// TIA Portal project "uMySQL_V0.3" (V15.1)

(* hardware
DEVICE "S7-1200 station_1"  S7-1200 Station
   slot 0: "Rack_0"  S7-1200 Rack  Rack  V1.0
   slot 1: "PLC_1"  CPU 1215C DC/DC/DC  6ES7 215-1AG40-0XB0  V4.2
*)

// ===== PLC "PLC_1"  CPU 1215C DC/DC/DC =====

VAR_GLOBAL   // PLC tag table "默认变量表"
   "Tag_1" AT %M100.0 : Bool;
   "Tag_2" AT %M100.1 : Bool;
   "Tag_3" AT %M100.2 : Bool;
END_VAR

TYPE "uMySQL_CDD"
   STRUCT
      Connect_OK : Bool;
      Connect_ID : Conn_Ouc;
      Connect_Sequence : DInt;
      Server_Protocol_Version : Int;
      Server_Server_Version : String;
      Server_Character_Set : Byte;
      CLIENT_PLUGIN_AUTH : String;
   END_STRUCT;
END_TYPE

DATA_BLOCK "uMySQL_Connect_DB"   // DB1
{ S7_Optimized_Access := 'TRUE' }
VERSION : 0.1
// stored: InstanceOfName uMySQL_Connect
"uMySQL_Connect"
BEGIN
   IP.RemoteAddress.ADDR[4] := 16#E0;
   IP.InterfaceId := 64;
   IP.ID := 16#65;
END_DATA_BLOCK

DATA_BLOCK "测试数据块"   // DB2
{ S7_Optimized_Access := 'TRUE' }
VERSION : 0.1
   VAR
      wstring : WString[2048];
      ad : Array[0..2048] of Byte;
   END_VAR
BEGIN
END_DATA_BLOCK

DATA_BLOCK "uMySQL_Query_DB"   // DB3
{ S7_Optimized_Access := 'TRUE' }
VERSION : 0.1
// stored: InstanceOfName uMySQL_Query
"uMySQL_Query"
BEGIN
END_DATA_BLOCK

DATA_BLOCK "uMySQL_Query_DB_1"   // DB4
{ S7_Optimized_Access := 'TRUE' }
VERSION : 0.1
// stored: InstanceOfName uMySQL_Query
"uMySQL_Query"
BEGIN
END_DATA_BLOCK

DATA_BLOCK "uMySQL_INI_DB_DB"   // DB5
{ S7_Optimized_Access := 'TRUE' }
VERSION : 0.1
// stored: InstanceOfName uMySQL_INI_DB
"uMySQL_INI_DB"
BEGIN
END_DATA_BLOCK

ORGANIZATION_BLOCK "Main"   // OB1, LAD, ProgramCycle
TITLE = "Main Program Sweep (Cycle)"
{ S7_Optimized_Access := 'TRUE' }
VERSION : 0.1
   VAR_INPUT
      Initial_Call : Bool;   // Initial call of this OB
      Remanence : Bool;   // =True, if remanent data are available
   END_VAR
BEGIN

REGION Network 1
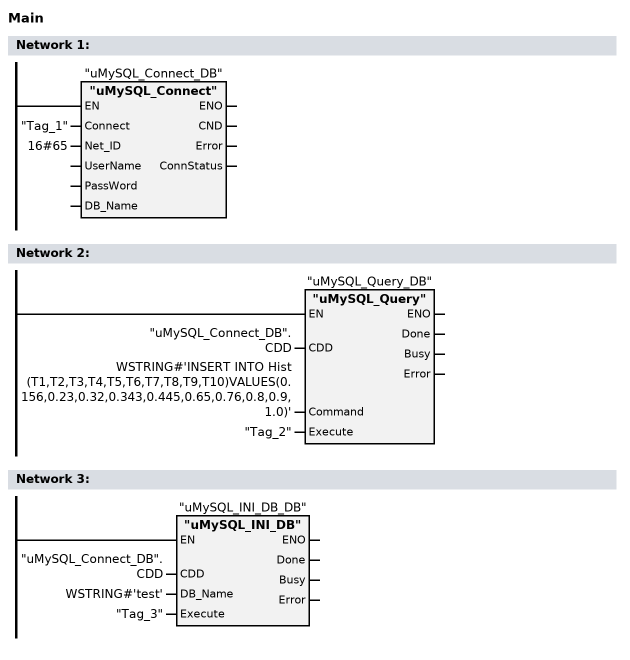
   RUNG wire#powerrail
      "uMySQL_Connect_DB"(Connect := "Tag_1", Net_ID := 16#65, UserName :=, PassWord :=, DB_Name :=, CND =>, Error =>, ConnStatus =>)
   END_RUNG
   // the same network as SCL:
   "uMySQL_Connect_DB"(Connect := "Tag_1", Net_ID := 16#65);   // "uMySQL_Connect"
END_REGION

REGION Network 2
   RUNG wire#powerrail
      "uMySQL_Query_DB"(CDD := "uMySQL_Connect_DB".CDD, Command := WSTRING#'INSERT INTO Hist (T1,T2,T3,T4,T5,T6,T7,T8,T9,T10)VALUES(0.156,0.23,0.32,0.343,0.445,0.65,0.76,0.8,0.9,1.0)', Execute := "Tag_2", Done =>, Busy =>, Error =>)
   END_RUNG
   // the same network as SCL:
   "uMySQL_Query_DB"(CDD := "uMySQL_Connect_DB".CDD,   // "uMySQL_Query"
                     Command := WSTRING#'INSERT INTO Hist (T1,T2,T3,T4,T5,T6,T7,T8,T9,T10)VALUES(0.156,0.23,0.32,0.343,0.445,0.65,0.76,0.8,0.9,1.0)',
                     Execute := "Tag_2");
END_REGION

REGION Network 3
   RUNG wire#powerrail
      "uMySQL_INI_DB_DB"(CDD := "uMySQL_Connect_DB".CDD, DB_Name := WSTRING#'test', Execute := "Tag_3", Done =>, Busy =>, Error =>)
   END_RUNG
   // the same network as SCL:
   "uMySQL_INI_DB_DB"(CDD := "uMySQL_Connect_DB".CDD, DB_Name := WSTRING#'test', Execute := "Tag_3");   // "uMySQL_INI_DB"
END_REGION
END_ORGANIZATION_BLOCK

// folder: uMySQL

FUNCTION_BLOCK "uMySQL_Connect"   // FB3, SCL
{ S7_Optimized_Access := 'TRUE' }
VERSION : 0.1
   VAR_INPUT
      Connect : Bool;   // True:发起连接；False:断开连接
      Net_ID : Conn_Ouc;   // 连接ID
      UserName : String := 'root';   // 数据库用户名
      PassWord : String := 'root';   // 数据库密码
      DB_Name : String := 'hist';   // 数据库名
   END_VAR
   VAR_OUTPUT
      CND : Bool;
      Error : Bool;
      ConnStatus : Byte;
   END_VAR
   VAR
      IP : TCON_IP_v4;
      CDD : "uMySQL_CDD";   // 共用的数据库连接参数
      TempBool : Array[0..19] of Bool;
      REV_Buffer : Array[0..#MessageMaxLen] of Byte;
      SND_Buffer : Array[0..#MessageMaxLen] of Byte;
      NetConnect : TCON;
      NetRcv : TRCV;
      NetRcv_EN : Bool;
      NetRcv_Len : Int;
      NetRcv_Done : Bool;
      "Step" : Int;
      MessageLen : Int;   // 消息帧长度
      SaltLen : Int;   // 挑战随机数长度
      Server_Auth_PlugIn_Name : String;
      ServerVersion_StartNum : Int;
      ServerCapability_flag : DWord;
      SaltString : Array[0..49] of Byte;
      Client_CapabilityFlag : DWord := 16#8609;   // 客户端权能标志位
      Client_MaxLen : DWord;
      Calc_Encryption_SHA1 : "Calc_Encryption_SHA1";
      Temp_SHA1 : Array[0..19] of Byte;
      Temp_SHA_Arry : Array[0..55] of Byte;
      Temp_SHA_Arry_Num : UInt;
      Temp_SHA_Arry_Num_Int : Int;
      Temp_SHA1_2 : Array[0..19] of Byte;
      Temp_SHA1_3 : Array[0..19] of Byte;
      Token : Array[0..19] of Byte;
      NetDISCON : TDISCON;
      NetDiscon_EN : Bool;
      NetSend : TSEND;
      NetSend_EN : Bool;
      NetSend_Done : Bool;
      TDiag_Result : TDiag_Status;
      NetDiag : T_DIAG;
      NetDiag_EN : Bool;
      NetSendLen : Int;
      Timer_ON : TON_TIME;
      Timer_OFF : TON_TIME;
      Timer_Error : TON_TIME;
      NetSendEnd : TSEND;
      NetSendEnd_EN : Bool;
      NetSendEnd_Done : Bool;
   END_VAR
   VAR_TEMP
      Temp_Dword : DWord;
      Temp_Index_i : Int;
      Temp_NowNum : Int;
      Temp_StrLen : Int;
   END_VAR
   VAR CONSTANT
      MessageMaxLen : DInt := 2048;   // 收发消息的最大长度
   END_VAR
   // IP.RemotePort := 3306;
   // IP.RemoteAddress.ADDR[4] := 16#A8;
   // IP.RemoteAddress.ADDR[3] := 16#1F;
   // IP.RemoteAddress.ADDR[2] := 16#A8;
   // IP.RemoteAddress.ADDR[1] := 16#C0;
   // IP.ActiveEstablished := true;
   // // CDD.Connect_OK : 数据库是否连接状态True:已连接；False :未连接
   // // CDD.Connect_ID : 连接ID，用于传递
   // // CDD.Connect_Sequence : 命令Sequence，用于传递
BEGIN


   (***********************************************************初始化数据******************************************************************)
   IF #Connect AND  #TempBool[0]=FALSE THEN
       #TempBool[0] := TRUE;
       #TempBool[1] := FALSE;
       #Step := 0;
       #CDD.Connect_ID := #Net_ID;
       #IP.ID := #Net_ID;
       #NetRcv_EN := TRUE;
       #NetDiscon_EN := FALSE;
       #NetSendEnd_EN := FALSE;
       ;
   END_IF;
   (***********************************************************断开连接******************************************************************)
   IF #Connect = FALSE AND #TempBool[1]=FALSE THEN
       #TempBool[0] := FALSE;
       #TempBool[1] := TRUE;
       #Step := 6;
   END_IF;


   #NetConnect(REQ:=#Connect,
               ID:=  #CDD.Connect_ID,
               CONNECT:=#IP);
   #NetRcv(EN_R:=#NetRcv_EN,
           ID:=#CDD.Connect_ID,
           LEN:=0,
           ADHOC:=TRUE,
           DATA:=#REV_Buffer);
   IF #NetRcv.NDR THEN
       #NetRcv_Done := TRUE;
   END_IF;
   (***********************************************************处理流程******************************************************************)
   //#Step 0  发起连接
   //#Step 1 等待MySQL服务器发回来的数据
   //#Step 2 解码发回来的认证数据，并计算需要响应的数据放入Sendbuffer
   //#Step 3 开始发送并等待发送完成
   //#Step 4 发送完成等待返回认证结果
   //#Step 5 解析返回结果是否已经连接成功
   //#Step 6 申请断开连接

   CASE #Step OF
       0:  // 如果在等待服务器第一次连接
           IF #NetConnect.DONE THEN
               #Step := 1;
           END_IF;
       1:  // 连接并等待返回第一次握手数据
           IF     #NetRcv_Done  THEN
               #NetRcv_Done := FALSE;
               #Step := 2;
               #NetRcv_EN := FALSE;
               #NetRcv_Len := UDINT_TO_INT(#NetRcv.RCVD_LEN);
           END_IF;
       2:
           REGION MySQL_Auth_Packet
               #Temp_Dword.%B0 := #REV_Buffer[0];
               #Temp_Dword.%B1 := #REV_Buffer[1];
               #Temp_Dword.%B2 := #REV_Buffer[2];
               #Temp_Dword.%B3 := b#16#00;
               #MessageLen := DINT_TO_INT(DWORD_TO_DINT(#Temp_Dword)); //实际传输数据的字符长度
               #CDD.Connect_Sequence := BYTE_TO_INT(#REV_Buffer[3]); //传输的Sequence值

               #CDD.Server_Protocol_Version := BYTE_TO_INT(#REV_Buffer[4]); //MySQL服务器的协议版本号，当前大多为10(16#0A)
               #ServerVersion_StartNum := 5;
               WHILE #REV_Buffer[#ServerVersion_StartNum] <> b#16#00 DO//MySQL服务器的版本号，第5个字符开始，00结尾
                   #CDD.Server_Server_Version[#ServerVersion_StartNum-4] := #REV_Buffer[#ServerVersion_StartNum];
                   #ServerVersion_StartNum := #ServerVersion_StartNum + 1;
               END_WHILE;
               #ServerVersion_StartNum := #ServerVersion_StartNum + 1;//b#16#00是服务器版本号的结尾，要跳到下一个字节
               #ServerVersion_StartNum := #ServerVersion_StartNum + 4;//跳过服务器线程ID

               FOR #Temp_Index_i := 0 TO 7 DO
                   #SaltString[#Temp_Index_i] := #REV_Buffer[#ServerVersion_StartNum];//挑战字符串的前8个Byte
                   #ServerVersion_StartNum := #ServerVersion_StartNum + 1;
               END_FOR;
               #ServerVersion_StartNum := #ServerVersion_StartNum + 1;
               #ServerCapability_flag.%B3 := #REV_Buffer[#ServerVersion_StartNum];//权能标志位低-低字节
               #ServerVersion_StartNum := #ServerVersion_StartNum + 1;
               #ServerCapability_flag.%B2 := #REV_Buffer[#ServerVersion_StartNum];//权能标志位低-高字节
               #ServerVersion_StartNum := #ServerVersion_StartNum + 1;
               #CDD.Server_Character_Set := #REV_Buffer[#ServerVersion_StartNum]; //采用字符集
               #ServerVersion_StartNum := #ServerVersion_StartNum + 1;
               #ServerVersion_StartNum := #ServerVersion_StartNum + 2;
               #ServerCapability_flag.%B1 := #REV_Buffer[#ServerVersion_StartNum];//权能标志位高-低字节
               #ServerVersion_StartNum := #ServerVersion_StartNum + 1;
               #ServerCapability_flag.%B0 := #REV_Buffer[#ServerVersion_StartNum];//权能标志位高-高字节
               #ServerVersion_StartNum := #ServerVersion_StartNum + 1;
               #SaltLen := BYTE_TO_INT(#REV_Buffer[#ServerVersion_StartNum]) -1; //采用挑战随机数的数量
               #ServerVersion_StartNum := #ServerVersion_StartNum + 1;
               #ServerVersion_StartNum := #ServerVersion_StartNum + 10;//跳过保留的10个B#16#00
               FOR #Temp_Index_i := 0 TO #SaltLen - 9 DO   //去掉前面的8个数据，同时从0开始，所以-9
                   #SaltString[#Temp_Index_i + 8] := #REV_Buffer[#ServerVersion_StartNum];//挑战字符串的后面N个Byte
                   #ServerVersion_StartNum := #ServerVersion_StartNum + 1;
               END_FOR;
               #ServerVersion_StartNum := #ServerVersion_StartNum + 1;
               #Temp_Index_i := 0;
               WHILE #REV_Buffer[#ServerVersion_StartNum] <> b#16#00 DO//MySQL服务器的版本号，第5个字符开始，00结尾
                   #CDD.CLIENT_PLUGIN_AUTH[#Temp_Index_i+1] := #REV_Buffer[#ServerVersion_StartNum];
                   #ServerVersion_StartNum := #ServerVersion_StartNum + 1;
                   #Temp_Index_i := #Temp_Index_i + 1;
               END_WHILE;

               (*
               FOR #Temp_Index_i := #ServerVersion_StartNum TO #MessageLen - 1 DO   //去掉前面的8个数据，同时从0开始，所以-9
                   #SaltString[#Temp_Index_i - #ServerVersion_StartNum + 2] := #REV_Buffer[#ServerVersion_StartNum];//挑战字符串的后面N个Byte
                   #ServerVersion_StartNum := #ServerVersion_StartNum + 1;
               END_FOR;*)
           END_REGION

           REGION Client_Auth_Packet
               #Temp_NowNum := 0;
               #Client_MaxLen := DINT_TO_DWORD(#MessageMaxLen);
               // Length                            3     Byte   最后处理
               #Temp_NowNum := #Temp_NowNum +3;
               // Sequence                      1     Byte
               #SND_Buffer[#Temp_NowNum] :=SINT_TO_BYTE( DINT_TO_SINT(#CDD.Connect_Sequence + 1));
               #Temp_NowNum := #Temp_NowNum + 1;
               // CapabilityFlag               4     Byte
               #SND_Buffer[#Temp_NowNum] := #Client_CapabilityFlag.%B0;
               #Temp_NowNum := #Temp_NowNum + 1;
               #SND_Buffer[#Temp_NowNum] := #Client_CapabilityFlag.%B1;
               #Temp_NowNum := #Temp_NowNum + 1;
               #SND_Buffer[#Temp_NowNum] := #Client_CapabilityFlag.%B2;
               #Temp_NowNum := #Temp_NowNum + 1;
               #SND_Buffer[#Temp_NowNum] := #Client_CapabilityFlag.%B3;
               #Temp_NowNum := #Temp_NowNum + 1;
               // Max_Length                   4     Byte
               #SND_Buffer[#Temp_NowNum] := #Client_MaxLen.%B0;
               #Temp_NowNum := #Temp_NowNum + 1;
               #SND_Buffer[#Temp_NowNum] := #Client_MaxLen.%B1;
               #Temp_NowNum := #Temp_NowNum + 1;
               #SND_Buffer[#Temp_NowNum] := #Client_MaxLen.%B2;
               #Temp_NowNum := #Temp_NowNum + 1;
               #SND_Buffer[#Temp_NowNum] := #Client_MaxLen.%B3;
               #Temp_NowNum := #Temp_NowNum + 1;
               // CharacterSet                 1     Byte
               #SND_Buffer[#Temp_NowNum] := #CDD.Server_Character_Set;
               #Temp_NowNum := #Temp_NowNum + 1;
               // Fill Data  (16#00)          23  Byte
               FOR #Temp_Index_i := 0 TO 22 DO
                   #SND_Buffer[#Temp_NowNum + #Temp_Index_i] := b#16#00;
               END_FOR;
               #Temp_NowNum := #Temp_NowNum + 23;
               // User Name                    N    Byte    Last Character    16#00
               #Temp_StrLen := LEN(#UserName);
               FOR #Temp_Index_i := 0 TO #Temp_StrLen - 1 DO
                   #SND_Buffer[#Temp_NowNum + #Temp_Index_i] := #UserName[#Temp_Index_i + 1];
               END_FOR;
               #Temp_NowNum := #Temp_NowNum + #Temp_StrLen;
               #SND_Buffer[#Temp_NowNum] := b#16#00;
               #Temp_NowNum := #Temp_NowNum + 1;
               #SND_Buffer[#Temp_NowNum] := b#16#14;
               #Temp_NowNum := #Temp_NowNum + 1;
               // Token                              N    Byte    Last Character    16#00
               #Calc_Encryption_SHA1(IN_Str := #PassWord,
                                     TempOutStr => #Temp_SHA1);
               #Calc_Encryption_SHA1(IN_Str := #Temp_SHA1,
                                     Len:=20,
                                     TempOutStr => #Temp_SHA1_2);
               // Strg_TO_Chars(Strg := #PassWord,
               //               pChars := 0,
               //               Cnt => #Temp_SHA_Arry_Num,
               //               Chars := #Temp_SHA_Arry);
               // #Temp_SHA_Arry_Num_Int := UINT_TO_INT(#Temp_SHA_Arry_Num);

               FOR #Temp_Index_i := 0 TO 19 DO
                   #Temp_SHA_Arry[#Temp_Index_i] := #SaltString[#Temp_Index_i];
               END_FOR;
               FOR #Temp_Index_i := 20 TO 39 DO
                   #Temp_SHA_Arry[#Temp_Index_i] := #Temp_SHA1_2[#Temp_Index_i - 20];
               END_FOR;

               #Calc_Encryption_SHA1(IN_Str := #Temp_SHA_Arry,
                                     Len := 40,
                                     TempOutStr => #Temp_SHA1_3);

               FOR #Temp_Index_i := 0 TO 19 DO
                   #Token[#Temp_Index_i] := #Temp_SHA1[#Temp_Index_i] XOR #Temp_SHA1_3[#Temp_Index_i];
                   #SND_Buffer[#Temp_NowNum + #Temp_Index_i] := #Token[#Temp_Index_i];
               END_FOR;
               #Temp_NowNum := #Temp_NowNum + 20;
               #SND_Buffer[#Temp_NowNum] := b#16#00;
               #Temp_NowNum := #Temp_NowNum + 1;

               // DataBase Name           N    Byte    Last Character    16#00
               #Temp_StrLen := LEN(#DB_Name);
               FOR #Temp_Index_i := 0 TO #Temp_StrLen - 1 DO
                   #SND_Buffer[#Temp_NowNum + #Temp_Index_i] := #DB_Name[#Temp_Index_i + 1];
               END_FOR;
               #Temp_NowNum := #Temp_NowNum + #Temp_StrLen;
               #SND_Buffer[#Temp_NowNum] := b#16#00;
               #Temp_NowNum := #Temp_NowNum + 1;
               //CLIENT_PLUGIN_AUTH
               #Temp_StrLen := LEN(#CDD.CLIENT_PLUGIN_AUTH);
               FOR #Temp_Index_i := 0 TO #Temp_StrLen - 1 DO
                   #SND_Buffer[#Temp_NowNum + #Temp_Index_i] := #CDD.CLIENT_PLUGIN_AUTH[#Temp_Index_i + 1];
               END_FOR;
               #Temp_NowNum := #Temp_NowNum + #Temp_StrLen;
               #SND_Buffer[#Temp_NowNum] := b#16#00;
               #Temp_NowNum := #Temp_NowNum + 1;

               //数据长度写入前三个byte
               #Temp_Dword := DINT_TO_DWORD(INT_TO_DINT(#Temp_NowNum - 4));
               #SND_Buffer[0] := #Temp_Dword.%B0;
               #SND_Buffer[1] := #Temp_Dword.%B1;
               #SND_Buffer[2] := #Temp_Dword.%B2;
               #Step := 3;
               #NetSendLen := #Temp_NowNum;
           END_REGION

           ;

       3:  // 等待发送完成
           #NetRcv_EN := TRUE;
           #NetSend_EN := TRUE;
           IF #NetSend_Done THEN
               #NetSend_Done := FALSE;
               #NetSend_EN := FALSE;
               #Step := 4;
           END_IF;

       4:  // 等待接收数据

           IF    #NetRcv_Done  THEN
               #NetRcv_Done := FALSE;

               #NetRcv_Len := UDINT_TO_INT(#NetRcv.RCVD_LEN);
               #NetRcv_EN := FALSE;
               #Step := 5;
           END_IF;
       5:  // 如果在等待服务器第一次连接
           IF #REV_Buffer[5]=b#16#00 AND  #NetRcv_Len >7 THEN
               #CND := TRUE;
           END_IF;


       6:  // 申请服务器断开连接
            #SND_Buffer[0] := b#16#01;
            #SND_Buffer[1] := b#16#00;
            #SND_Buffer[2] := b#16#00;
            #SND_Buffer[3] := b#16#00;
            #SND_Buffer[4] := b#16#01;
            #NetSendEnd_EN := TRUE;
            IF #NetSendEnd_Done THEN
                #Step := 7;
            END_IF;

        7:  // 申请服务器断开连接

            #NetDiscon_EN := TRUE;
        8:
            ;
       ELSE  // Statement section ELSE
           ;
   END_CASE;
   (***********************************************************发送数据******************************************************************)
   #NetSend(REQ := #NetSend_EN,
            ID := #Net_ID,
           // DONE=>#NetSend_Done,
            LEN :=INT_TO_UDINT(#NetSendLen),// INT_TO_UINT(#Temp_NowNum),
            DATA := #SND_Buffer);
   IF #NetSend.DONE THEN
       #NetSend_Done := TRUE;
   END_IF;

   #NetSendEnd(REQ:=#NetSendEnd_EN,
               ID:=#Net_ID,
               LEN:=5,
               DONE=>#NetSendEnd_Done,
               DATA:=#SND_Buffer);





   (***********************************************************断开连接******************************************************************)

   #NetDISCON(REQ:=#NetDiscon_EN AND #Timer_ON.Q ,
              ID:=#Net_ID);

   #Timer_ON(IN := NOT #Timer_OFF.Q,
             PT := t#0.5s);

   #Timer_OFF(IN := #Timer_ON.Q,
              PT := t#0.5s);




   (***********************************************************监测连接******************************************************************)
   #NetDiag(REQ := #Timer_ON.Q,
            ID := #Net_ID,
            RESULT := #TDiag_Result);
   IF  #NetDiag.ERROR THEN
       #ConnStatus := B#16#00;
   END_IF;
   IF #NetDiag.DONE THEN
       #ConnStatus := #TDiag_Result.State;
   END_IF;
   IF #ConnStatus <> B#16#04 THEN
       #CND := FALSE;
   END_IF;

   #CDD.Connect_OK := #CND;

   #Timer_Error(IN:=#Connect AND NOT #CND,
                PT:=t#3s);

   #Error := #Timer_Error.Q;
END_FUNCTION_BLOCK

FUNCTION_BLOCK "uMySQL_Query"   // FB5, SCL
{ S7_Optimized_Access := 'TRUE' }
VERSION : 0.1
   VAR_INPUT
      CDD : "uMySQL_CDD";
      Command : WString[2048];
      Execute : Bool;
   END_VAR
   VAR_OUTPUT
      Done : Bool;
      Busy : Bool;
      Error : Bool;
   END_VAR
   VAR
      Net_Send : TSEND;
      Net_Send_EN : Bool;
      Net_Send_Done : Bool;
      Net_Send_Len : UInt;
      Command_Len : UInt;
      Net_Recv : TRCV;
      Net_Recv_EN : Bool;
      Net_Recv_Done : Bool;
      Net_Recv_Len : UInt;
      Temp_Bool : Array[0..19] of Bool;
      SendBuffer : Array[0..2048] of Byte;
      RecvBuffer : Array[0..2048] of Byte;
      SendBufferWChar : Array[0..2048] of WChar;
      TRCV : TRCV;
   END_VAR
   VAR_TEMP
      Temp_Index_i : Int;
      Temp_Dword : DWord;
   END_VAR
BEGIN

   IF #Execute THEN
      // #Net_Recv_EN := TRUE;
      ;
   END_IF;

   IF #Execute AND NOT #Temp_Bool[0] THEN
       #Temp_Bool[0] := TRUE;
       #Net_Send_EN := TRUE;
       #Command_Len :=INT_TO_UINT( LEN(#Command));
       #SendBuffer[4] := B#16#03;

       Strg_TO_Chars(Strg := #Command,
                     pChars := 0,
                     Cnt => #Command_Len,
                     Chars := #SendBufferWChar);

       FOR #Temp_Index_i := 0 TO UINT_TO_INT( #Command_Len) -1 DO
           #SendBuffer[#Temp_Index_i + 5]:=WCHAR_TO_BYTE(#SendBufferWChar[#Temp_Index_i]) ;
       END_FOR;
       #Net_Send_Len :=#Command_Len + 5;
       #Net_Send_EN := TRUE;
       //数据长度写入前三个byte
       #Temp_Dword := DINT_TO_DWORD(INT_TO_DINT(UINT_TO_INT(#Net_Send_Len) - 4));
       #SendBuffer[0] := #Temp_Dword.%B0;
       #SendBuffer[1] := #Temp_Dword.%B1;
       #SendBuffer[2] := #Temp_Dword.%B2;
   END_IF;


   IF NOT #Execute THEN
       #Temp_Bool[0] := FALSE;
       #Net_Recv_Len := 0;
       #Net_Recv_Done := FALSE;
       #Net_Send_EN := FALSE;
       #Net_Recv_EN := FALSE;
   END_IF;


   #Net_Send(REQ:=#Net_Send_EN,
             ID:=#CDD.Connect_ID,
             LEN:=#Net_Send_Len,
             DONE=>#Net_Send_Done,
             DATA:=#SendBuffer);

   IF #Net_Send.DONE OR #Net_Send.ERROR THEN
       #Net_Send_EN := FALSE;
   END_IF;

   // #Net_Recv(EN_R:=#Net_Recv_EN,
   //           ID:=#CDD.Connect_ID,
   //           LEN:=0,
   //           ADHOC:=TRUE,
   //           NDR=>#Net_Recv_Done,
   //           DATA:=#Net_Recv);




   IF #Net_Recv.NDR THEN
       #Net_Recv_Len := UDINT_TO_UINT(#Net_Recv.RCVD_LEN);
       #Net_Recv_Done := TRUE;
   END_IF;
END_FUNCTION_BLOCK

FUNCTION_BLOCK "Calc_Encryption_SHA1"   // FB6, SCL
{ S7_Optimized_Access := 'FALSE' }
VERSION : 0.1
   VAR_INPUT
      IN_Str : Variant;
      Len : Int;
   END_VAR
   VAR_OUTPUT
      TempOutStr : Array[0..19] of Byte;
      Encrption AT TempOutStr : Array[0..4] of DWord;
   END_VAR
   VAR_TEMP
      "A" : DWord;
      "B" : DWord;
      C : DWord;
      D : DWord;
      "E" : DWord;
      Length : Int;
      Lenth_Uint : UInt;
      MessageBlock : Array[0..63] of Byte;
      MessageBlock_DWORD AT MessageBlock : Array[0..15] of DWord;
      W : Array[0..79] of DWord;
      Index_i : Int;
      temp : DWord;
      Temp_Str : String;
      Temp_Array : Array[0..446] of Byte;
   END_VAR
   VAR CONSTANT
      K0 : DWord := 16#5A827999;   // K0计算常量
      K1 : DWord := 16#6ED9EBA1;   // K1计算常量
      K2 : DWord := 16#8F1BBCDC;   // K2计算常量
      K3 : DWord := 16#CA62C1D6;   // K3计算常量
      Const_A : DWord := 16#67452301;   // 链接变量A
      Const_B : DWord := 16#EFCDAB89;   // 链接变量B
      Const_C : DWord := 16#98BADCFE;   // 链接变量C
      Const_D : DWord := 16#10325476;   // 链接变量D
      Const_E : DWord := 16#C3D2E1F0;   // 链接变量E
   END_VAR
BEGIN
   (***************************************************数据初始化******************************************************)
   #A := #Const_A;
   #B := #Const_B;
   #C := #Const_C;
   #D := #Const_D;
   #E := #Const_E;
   //#Length := LEN(#IN_Str);
   FILL_BLK(IN := B#16#00,  COUNT := 64,  OUT => #MessageBlock[0]);
   FILL_BLK(IN := DW#16#000000000,   COUNT := 80,  OUT => #W[0]);




   (*************************************************填充/准备数据****************************************************)
   IF TypeOf(#IN_Str) =String THEN
       //如果是字符串
       VariantGet(SRC:=#IN_Str,
                  DST=>#Temp_Str);
       #Length := LEN(#Temp_Str);

       Strg_TO_Chars(Strg :=#Temp_Str ,
                     pChars := 0,
                     Cnt => #Lenth_Uint,
                     Chars := #MessageBlock);   //填充客户输入字符
   ELSE
       IF IS_ARRAY(#IN_Str) THEN
          // #Length:=UDINT_TO_INT(CountOfElements(#IN_Str)) ;
           #Length := #Len;
           VariantGet(SRC:=#IN_Str,     DST=>#Temp_Array);
           MOVE_BLK(IN := #Temp_Array[0],  COUNT :=INT_TO_UINT( #Length),  OUT => #MessageBlock[0]);
       END_IF;
     ;
   END_IF;
   (*********************************************输入数据安全检测****************************************************)
   IF (#Length = 0) OR (#Length > 56) THEN
       RETURN;
   END_IF;

   #MessageBlock[#Length] := B#16#80;   //后一位填1，其他全为0
   #MessageBlock_DWORD[14] :=DW#16#00000000;          //填充数据长度高位
   #MessageBlock_DWORD[15] := DINT_TO_DWORD(#Length * 8);//填充数据长度低位
   MOVE_BLK(IN := #MessageBlock_DWORD[0],  COUNT := 16,  OUT => #W[0]);
   FOR #Index_i := 16 TO 79 DO
       #W[#Index_i] := ROL(N := 1, IN := (#W[#Index_i - 3] XOR #W[#Index_i - 8] XOR #W[#Index_i - 14] XOR #W[#Index_i - 16]));
   END_FOR;
   (*************************************************计算过程****************************************************)
   FOR #Index_i := 0 TO 19 DO
       #temp := ROL(IN := #A, N := 5) + ((#B AND #C) OR (NOT (#B) AND #D)) + #E + #W[#Index_i] + #K0;
       #E := #D;
       #D := #C;
       #C := ROL(IN := #B, N := 30);
       #B := #A;
       #A := #temp;
   END_FOR;

   FOR #Index_i := 20 TO 39 DO
       #temp := ROL(IN := #A, N := 5) + (#B XOR #C XOR #D) + #E + #W[#Index_i] + #K1;
       #E := #D;
       #D := #C;
       #C := ROL(N := 30, IN := #B);
       #B := #A;
       #A := #temp;
   END_FOR;

   FOR #Index_i := 40 TO 59 DO
       #temp := ROL(N := 5, IN := #A) + ((#B AND #C) OR (#B AND #D) OR (#C AND #D)) + #E + #W[#Index_i] + #K2;
       #E := #D;
       #D := #C;
       #C := ROL(N := 30, IN := #B);
       #B := #A;
       #A := #temp;
   END_FOR;

   FOR #Index_i := 60 TO 79 DO
       #temp := ROL(N := 5, IN := #A) + (#B XOR #C XOR #D) + #E + #W[#Index_i] + #K3;
       #E := #D;
       #D := #C;
       #C := ROL(N := 30, IN := #B);
       #B := #A;
       #A := #temp;
   END_FOR;

   #Encrption[0] := #Const_A + #A;
   #Encrption[1] := #Const_B+ #B;
   #Encrption[2] := #Const_C + #C;
   #Encrption[3] := #Const_D + #D;
   #Encrption[4] := #Const_E + #E;
END_FUNCTION_BLOCK

FUNCTION_BLOCK "uMySQL_INI_DB"   // FB7, SCL
{ S7_Optimized_Access := 'TRUE' }
VERSION : 0.1
   VAR_INPUT
      CDD : "uMySQL_CDD";
      DB_Name : WString[2048];
      Execute : Bool;
   END_VAR
   VAR_OUTPUT
      Done : Bool;
      Busy : Bool;
      Error : Bool;
   END_VAR
   VAR
      Net_Send : TSEND;
      Net_Send_EN : Bool;
      Net_Send_Done : Bool;
      Net_Send_Len : UInt;
      Command_Len : UInt;
      Net_Recv : TRCV;
      Net_Recv_EN : Bool;
      Net_Recv_Done : Bool;
      Net_Recv_Len : UInt;
      Temp_Bool : Array[0..19] of Bool;
      SendBuffer : Array[0..2048] of Byte;
      RecvBuffer : Array[0..2048] of Byte;
      SendBufferWChar : Array[0..2048] of WChar;
   END_VAR
   VAR_TEMP
      Temp_Index_i : Int;
      Temp_Dword : DWord;
   END_VAR
BEGIN

   IF #Execute THEN
      // #Net_Recv_EN := TRUE;
      ;
   END_IF;

   IF #Execute AND NOT #Temp_Bool[0] THEN
       #Temp_Bool[0] := TRUE;
       #Net_Send_EN := TRUE;
       #Command_Len :=INT_TO_UINT( LEN(#DB_Name));
       #SendBuffer[4] := B#16#02;

       Strg_TO_Chars(Strg := #DB_Name,
                     pChars := 0,
                     Cnt => #Command_Len,
                     Chars := #SendBufferWChar);

       FOR #Temp_Index_i := 0 TO UINT_TO_INT( #Command_Len) -1 DO
           #SendBuffer[#Temp_Index_i + 5]:=WCHAR_TO_BYTE(#SendBufferWChar[#Temp_Index_i]) ;
       END_FOR;
       #Net_Send_Len :=#Command_Len + 5;
       #Net_Send_EN := TRUE;
       //数据长度写入前三个byte
       #Temp_Dword := DINT_TO_DWORD(INT_TO_DINT(UINT_TO_INT(#Net_Send_Len) - 4));
       #SendBuffer[0] := #Temp_Dword.%B0;
       #SendBuffer[1] := #Temp_Dword.%B1;
       #SendBuffer[2] := #Temp_Dword.%B2;
   END_IF;


   IF NOT #Execute THEN
       #Temp_Bool[0] := FALSE;
       #Net_Recv_Len := 0;
       #Net_Recv_Done := FALSE;
       #Net_Send_EN := FALSE;
       #Net_Recv_EN := FALSE;
   END_IF;


   #Net_Send(REQ:=#Net_Send_EN,
             ID:=#CDD.Connect_ID,
             LEN:=#Net_Send_Len,
             DONE=>#Net_Send_Done,
             DATA:=#SendBuffer);

   IF #Net_Send.DONE OR #Net_Send.ERROR THEN
       #Net_Send_EN := FALSE;
   END_IF;

   // #Net_Recv(EN_R:=#Net_Recv_EN,
   //           ID:=#CDD.Connect_ID,
   //           LEN:=0,
   //           ADHOC:=TRUE,
   //           NDR=>#Net_Recv_Done,
   //           DATA:=#Net_Recv);


   IF #Net_Recv.NDR THEN
       #Net_Recv_Len := UDINT_TO_UINT(#Net_Recv.RCVD_LEN);
       #Net_Recv_Done := TRUE;
   END_IF;
END_FUNCTION_BLOCK